TYPE ExampleComponents EXTENDS TcoCore.TcoStruct : 
STRUCT
    DmcReader : STRING;
    BoltPresenceSensor : BOOL;
    DimX_Sensor : LREAL;
    DimY_Sensor : LREAL;
    DimZ_Sensor : LREAL;
END_STRUCT
END_TYPE

(* stored: Version 1.1.0.1, ProductVersion 3.1.4024.9
   DUT ExampleComponents: Id {2b6326a9-8e03-0647-2962-aa10edbd1fa1} *)
